(* CODESYS project pwm_01.project

Project tree, tasks and I/O mapping:
  Device : MC4-26-20, Enovation Controls, order no. 58-70-0006, version 1.1.0.17
      input  batteryVoltage : Word  // Battery Voltage
      input  reg1Voltage : Word  // Regulator #1 Voltage
      input  reg2Voltage : Word  // Regulator #2 Voltage
      input  wakePinVoltage : Word  // Wake Pin Voltage
      input  sleepAllowed : BIT  // Sleep Allowed
      output enterSleep : BIT  // Enter Sleep
      input  bootReason : Byte  // Bootup Reason
      output userLED1State : BIT  // User LED 1 State
      output userLED2State : BIT  // User LED 2 State
      input  loadpwrVoltage : Word  // Load Power Voltage
      input  loadpwrProtected : Word  // Load Power Voltage (Protected)
      input  topRailTemp : Int  // Top Heatrail Temp
      input  botRailTemp : Int  // Bottom Heatrail Temp
      input  buildMajorVersion : BYTE  // Build Major Version
      input  buildMinorVersion : BYTE  // Build Minor Version
      input  buildPatchVersion : BYTE  // Build Patch Version
      input  firmwareMajorVersion : DWord  // Firmware Major Version
      input  firmwareMinorVersion : DWord  // Firmware Minor Version
      input  firmwareIdentifier : DWord  // Firmware Identifier
      input  serialNumber : DWord  // Serial Number
      input  hourMeter : Real  // Hour Meter
      input  startCount : DWord  // Cumulative Starts
      input  dynamicMemSize : UINT  // Dynamic Memory Size
      input  dynamicMemMaxUsage : UINT  // Dynamic Memory Max Usage
      input  relayCurrent : Real  // Relay Total Current
      input  relaySourcing : Real  // Relay Sourcing Current
      input  relaySinking : Real  // Relay Sinking Current
      output relayState : BIT  // Relay State
      input  relayIsActive : BIT  // Relay Active
      output clearActiveFaults : BIT  // Clear Active Faults (rising edge)
      input  activeFaultIsSet : BIT  // Active Fault Available
      input  activeFaultCount : UINT  // Active Fault Count
      output clearHistoricFaults : BIT  // Clear Historic Faults (rising edge)
      input  historicFaultIsSet : BIT  // Historic Fault Available
      input  historicFaultCount : UINT  // Historic Fault Count
      input  totalFaultCount : UINT  // Total Fault Count
      output fltMonIndex : UINT  // Fault Index
      input  fltMonIsEnabled : BIT  // Fault Is Enabled
      input  fltMonConditionPresent : BIT  // Fault Condition Present
      input  fltMonActive : BIT  // Fault Active Latched
      input  fltMonHistoric : BIT  // Fault Historic Latched
      input  fltMonCurrentStart : BIT  // Current start cycle
      input  fltMonActiveStarts : BYTE  // Starts since active
      output fltMonClearActive : BIT  // Clear Active (rising edge)
      output fltMonClearHistoric : BIT  // Clear Historic (rising edge)
      input  dcSwitchTemp : Int  // DC Switch Temp
      input  InputA04 : input_param_hi_spd_struct  // Input A04
      input  analogValueA04 : Real  // Input A04.Analog value
      input  digitalValueA04 : Bool  // Input A04.Digital value
      input  frequencyA04 : Word  // Input A04.Frequency
      input  dutyCycleA04 : Real  // Input A04.Duty cycle
      input  phaseAngleA04 : Real  // Input A04.Phase angle
      input  pulseCountA04 : DWord  // Input A04.Pulse count
      input  upDownCountA04 : DInt  // Input A04.Up/Down count
      input  freqHPA04 : Real  // Input A04.Frequency (high precision)
      input  freqTSA04 : Real  // Input A04.Frequency edge timestamp
      input  InputA05 : input_param_hi_spd_struct  // Input A05
      input  analogValueA05 : Real  // Input A05.Analog value
      input  digitalValueA05 : Bool  // Input A05.Digital value
      input  frequencyA05 : Word  // Input A05.Frequency
      input  dutyCycleA05 : Real  // Input A05.Duty cycle
      input  phaseAngleA05 : Real  // Input A05.Phase angle
      input  pulseCountA05 : DWord  // Input A05.Pulse count
      input  upDownCountA05 : DInt  // Input A05.Up/Down count
      input  freqHPA05 : Real  // Input A05.Frequency (high precision)
      input  freqTSA05 : Real  // Input A05.Frequency edge timestamp
      input  InputA07 : input_param_hi_spd_struct  // Input A07
      input  analogValueA07 : Real  // Input A07.Analog value
      input  digitalValueA07 : Bool  // Input A07.Digital value
      input  frequencyA07 : Word  // Input A07.Frequency
      input  dutyCycleA07 : Real  // Input A07.Duty cycle
      input  phaseAngleA07 : Real  // Input A07.Phase angle
      input  pulseCountA07 : DWord  // Input A07.Pulse count
      input  upDownCountA07 : DInt  // Input A07.Up/Down count
      input  freqHPA07 : Real  // Input A07.Frequency (high precision)
      input  freqTSA07 : Real  // Input A07.Frequency edge timestamp
      input  InputA10 : input_param_hi_spd_struct  // Input A10
      input  analogValueA10 : Real  // Input A10.Analog value
      input  digitalValueA10 : Bool  // Input A10.Digital value
      input  frequencyA10 : Word  // Input A10.Frequency
      input  dutyCycleA10 : Real  // Input A10.Duty cycle
      input  phaseAngleA10 : Real  // Input A10.Phase angle
      input  pulseCountA10 : DWord  // Input A10.Pulse count
      input  upDownCountA10 : DInt  // Input A10.Up/Down count
      input  freqHPA10 : Real  // Input A10.Frequency (high precision)
      input  freqTSA10 : Real  // Input A10.Frequency edge timestamp
      input  InputA11 : input_param_hi_spd_struct  // Input A11
      input  analogValueA11 : Real  // Input A11.Analog value
      input  digitalValueA11 : Bool  // Input A11.Digital value
      input  frequencyA11 : Word  // Input A11.Frequency
      input  dutyCycleA11 : Real  // Input A11.Duty cycle
      input  phaseAngleA11 : Real  // Input A11.Phase angle
      input  pulseCountA11 : DWord  // Input A11.Pulse count
      input  upDownCountyA11 : DInt  // Input A11.Up/Down count
      input  freqHPA11 : Real  // Input A11.Frequency (high precision)
      input  freqTSA11 : Real  // Input A11.Frequency edge timestamp
      input  InputA12 : input_param_hi_spd_struct  // Input A12
      input  analogValueA12 : Real  // Input A12.Analog value
      input  digitalValueA12 : Bool  // Input A12.Digital value
      input  frequencyA12 : Word  // Input A12.Frequency
      input  dutyCycleA12 : Real  // Input A12.Duty cycle
      input  phaseAngleA12 : Real  // Input A12.Phase angle
      input  pulseCountA12 : DWord  // Input A12.Pulse count
      input  upDownCountA12 : DInt  // Input A12.Up/Down count
      input  freqHPA12 : Real  // Input A12.Frequency (high precision)
      input  freqTSA12 : Real  // Input A12.Frequency edge timestamp
      input  InputB07 : input_param_hi_spd_struct  // Input B07
      input  analogValueB07 : Real  // Input B07.Analog value
      input  digitalValueB07 : Bool  // Input B07.Digital value
      input  frequencyB07 : Word  // Input B07.Frequency
      input  dutyCycleB07 : Real  // Input B07.Duty cycle
      input  phaseAngleB07 : Real  // Input B07.Phase angle
      input  pulseCountB07 : DWord  // Input B07.Pulse count
      input  upDownCountB07 : DInt  // Input B07.Up/Down count
      input  freqHPB07 : Real  // Input B07.Frequency (high precision)
      input  freqTSB07 : Real  // Input B07.Frequency edge timestamp
      input  InputB08 : input_param_hi_spd_struct  // Input B08
      input  analogValueB08 : Real  // Input B08.Analog value
      input  digitalValueB08 : Bool  // Input B08.Digital value
      input  frequencyB08 : Word  // Input B08.Frequency
      input  dutyCycleB08 : Real  // Input B08.Duty cycle
      input  phaseAngleB08 : Real  // Input B08.Phase angle
      input  pulseCountB08 : DWord  // Input B08.Pulse count
      input  upDownCountB08 : DInt  // Input B08.Up/Down count
      input  freqHPB08 : Real  // Input B08.Frequency (high precision)
      input  freqTSB08 : Real  // Input B08.Frequency edge timestamp
      input  InputB09 : input_param_hi_spd_struct  // Input B09
      input  analogValueB09 : Real  // Input B09.Analog value
      input  digitalValueB09 : Bool  // Input B09.Digital value
      input  frequencyB09 : Word  // Input B09.Frequency
      input  dutyCycleB09 : Real  // Input B09.Duty cycle
      input  phaseAngleB09 : Real  // Input B09.Phase angle
      input  pulseCountB09 : DWord  // Input B09.Pulse count
      input  upDownCountB09 : DInt  // Input B09.Up/Down count
      input  freqHPB09 : Real  // Input B09.Frequency (high precision)
      input  freqTSB09 : Real  // Input B09.Frequency edge timestamp
      input  InputB10 : input_param_hi_spd_struct  // Input B10
      input  analogValueB10 : Real  // Input B10.Analog value
      input  digitalValueB10 : Bool  // Input B10.Digital value
      input  frequencyB10 : Word  // Input B10.Frequency
      input  dutyCycleB10 : Real  // Input B10.Duty cycle
      input  phaseAngleB10 : Real  // Input B10.Phase angle
      input  pulseCountB10 : DWord  // Input B10.Pulse count
      input  upDownCountB10 : DInt  // Input B10.Up/Down count
      input  freqHPB10 : Real  // Input B10.Frequency (high precision)
      input  freqTSB10 : Real  // Input B10.Frequency edge timestamp
      input  InputA06 : input_param_struct  // Input A06
      input  analogValueA06 : Real  // Input A06.Analog value
      input  digitalValueA06 : Bool  // Input A06.Digital value
      input  frequencyA06 : Word  // Input A06.Frequency
      input  pulseCountA06 : DWord  // Input A06.Pulse count
      input  freqHPA06 : Real  // Input A06.Frequency (high precision)
      input  freqTSA06 : Real  // Input A06.Frequency edge timestamp
      input  InputA14 : input_param_struct  // Input A14
      input  analogValueA14 : Real  // Input A14.Analog value
      input  digitalValueA14 : Bool  // Input A14.Digital value
      input  frequencyA14 : Word  // Input A14.Frequency
      input  pulseCountA14 : DWord  // Input A14.Pulse count
      input  freqHPA14 : Real  // Input A14.Frequency (high precision)
      input  freqTSA14 : Real  // Input A14.Frequency edge timestamp
      input  InputA15 : input_param_struct  // Input A15
      input  analogValueA15 : Real  // Input A15.Analog value
      input  digitalValueA15 : Bool  // Input A15.Digital value
      input  frequencyA15 : Word  // Input A15.Frequency
      input  pulseCountA15 : DWord  // Input A15.Pulse count
      input  freqHPA15 : Real  // Input A15.Frequency (high precision)
      input  freqTSA15 : Real  // Input A15.Frequency edge timestamp
      input  InputA16 : input_param_struct  // Input A16
      input  analogValueA16 : Real  // Input A16.Analog value
      input  digitalValueA16 : Bool  // Input A16.Digital value
      input  frequencyA16 : Word  // Input A16.Frequency
      input  pulseCountA16 : DWord  // Input A16.Pulse count
      input  freqHPA16 : Real  // Input A16.Frequency (high precision)
      input  freqTSA16 : Real  // Input A16.Frequency edge timestamp
      input  InputA17 : input_param_struct  // Input A17
      input  analogValueA17 : Real  // Input A17.Analog value
      input  digitalValueA17 : Bool  // Input A17.Digital value
      input  frequencyA17 : Word  // Input A17.Frequency
      input  pulseCountA17 : DWord  // Input A17.Pulse count
      input  freqHPA17 : Real  // Input A17.Frequency (high precision)
      input  freqTSA17 : Real  // Input A17.Frequency edge timestamp
      input  InputA18 : input_param_struct  // Input A18
      input  analogValueA18 : Real  // Input A18.Analog value
      input  digitalValueA18 : Bool  // Input A18.Digital value
      input  frequencyA18 : Word  // Input A18.Frequency
      input  pulseCountA18 : DWord  // Input A18.Pulse count
      input  freqHPA18 : Real  // Input A18.Frequency (high precision)
      input  freqTSA18 : Real  // Input A18.Frequency edge timestamp
      input  InputB01 : input_param_struct  // Input B01
      input  analogValueB01 : Real  // Input B01.Analog value
      input  digitalValueB01 : Bool  // Input B01.Digital value
      input  frequencyB01 : Word  // Input B01.Frequency
      input  pulseCountB01 : DWord  // Input B01.Pulse count
      input  freqHPB01 : Real  // Input B01.Frequency (high precision)
      input  freqTSB01 : Real  // Input B01.Frequency edge timestamp
      input  InputB11 : input_param_struct  // Input B11
      input  analogValueB11 : Real  // Input B11.Analog value
      input  digitalValueB11 : Bool  // Input B11.Digital value
      input  frequencyB11 : Word  // Input B11.Frequency
      input  pulseCountB11 : DWord  // Input B11.Pulse count
      input  freqHPB11 : Real  // Input B11.Frequency (high precision)
      input  freqTSB11 : Real  // Input B11.Frequency edge timestamp
      input  InputB12 : input_param_struct  // Input B12
      input  analogValueB12 : Real  // Input B12.Analog value
      input  digitalValueB12 : Bool  // Input B12.Digital value
      input  frequencyB12 : Word  // Input B12.Frequency
      input  pulseCountB12 : DWord  // Input B12.Pulse count
      input  freqHPB12 : Real  // Input B12.Frequency (high precision)
      input  freqTSB12 : Real  // Input B12.Frequency edge timestamp
      input  InputB13 : input_param_struct  // Input B13
      input  analogValueB13 : Real  // Input B13.Analog value
      input  digitalValueB13 : Bool  // Input B13.Digital value
      input  frequencyB13 : Word  // Input B13.Frequency
      input  pulseCountB13 : DWord  // Input B13.Pulse count
      input  freqHPB13 : Real  // Input B13.Frequency (high precision)
      input  freqTSB13 : Real  // Input B13.Frequency edge timestamp
      input  InputC07 : input_param_struct  // Input C07
      input  analogValueC07 : Real  // Input C07.Analog value
      input  digitalValueC07 : Bool  // Input C07.Digital value
      input  frequencyC07 : Word  // Input C07.Frequency
      input  pulseCountC07 : DWord  // Input C07.Pulse count
      input  freqHPC07 : Real  // Input C07.Frequency (high precision)
      input  freqTSC07 : Real  // Input C07.Frequency edge timestamp
      input  InputC08 : input_param_struct  // Input C08
      input  analogValueC08 : Real  // Input C08.Analog value
      input  digitalValueC08 : Bool  // Input C08.Digital value
      input  frequencyC08 : Word  // Input C08.Frequency
      input  pulseCountC08 : DWord  // Input C08.Pulse count
      input  freqHPC08 : Real  // Input C08.Frequency (high precision)
      input  freqTSC08 : Real  // Input C08.Frequency edge timestamp
      input  InputC09 : input_param_struct  // Input C09
      input  analogValueC09 : Real  // Input C09.Analog value
      input  digitalValueC09 : Bool  // Input C09.Digital value
      input  frequencyC09 : Word  // Input C09.Frequency
      input  pulseCountC09 : DWord  // Input C09.Pulse count
      input  freqHPC09 : Real  // Input C09.Frequency (high precision)
      input  freqTSC09 : Real  // Input C09.Frequency edge timestamp
      input  InputC10 : input_param_struct  // Input C10
      input  analogValueC10 : Real  // Input C10.Analog value
      input  digitalValueC10 : Bool  // Input C10.Digital value
      input  frequencyC10 : Word  // Input C10.Frequency
      input  pulseCountC10 : DWord  // Input C10.Pulse count
      input  freqHPC10 : Real  // Input C10.Frequency (high precision)
      input  freqTSC10 : Real  // Input C10.Frequency edge timestamp
      input  InputC11 : input_param_struct  // Input C11
      input  analogValueC11 : Real  // Input C11.Analog value
      input  digitalValueC11 : Bool  // Input C11.Digital value
      input  frequencyC11 : Word  // Input C11.Frequency
      input  pulseCountC11 : DWord  // Input C11.Pulse count
      input  freqHPC11 : Real  // Input C11.Frequency (high precision)
      input  freqTSC11 : Real  // Input C11.Frequency edge timestamp
      input  InputC12 : input_param_struct  // Input C12
      input  analogValueC12 : Real  // Input C12.Analog value
      input  digitalValueC12 : Bool  // Input C12.Digital value
      input  frequencyC12 : Word  // Input C12.Frequency
      input  pulseCountC12 : DWord  // Input C12.Pulse count
      input  freqHPC12 : Real  // Input C12.Frequency (high precision)
      input  freqTSC12 : Real  // Input C12.Frequency edge timestamp
      input  chanStateB02 : Byte  // Channel state
      input  chanStateB03 : Byte  // Channel state
      input  chanStateB04 : Byte  // Channel state
      input  chanStateB05 : Byte  // Channel state
      input  chanStateB06 : Byte  // Channel state
      input  chanStateB14 : Byte  // Channel state
      input  chanStateB15 : Byte  // Channel state
      input  chanStateB16 : Byte  // Channel state
      input  chanStateB17 : Byte  // Channel state
      input  chanStateB18 : Byte  // Channel state
      input  chanStateC02 : Byte  // Channel state
      input  chanStateC03 : Byte  // Channel state
      input  chanStateC04 : Byte  // Channel state
      input  chanStateC05 : Byte  // Channel state
      input  chanStateC06 : Byte  // Channel state
      input  chanStateC14 : Byte  // Channel state
      input  chanStateC15 : Byte  // Channel state
      input  chanStateC16 : Byte  // Channel state
      input  chanStateC17 : Byte  // Channel state
      input  chanStateC18 : Byte  // Channel state
      output desiredDutyB02 : Real  // Desired Duty Cycle
      output desiredDutyB03 : Real  // Desired Duty Cycle
      output desiredDutyB04 : Real  // Desired Duty Cycle
      output desiredDutyB05 : Real  // Desired Duty Cycle
      output desiredDutyB06 : Real  // Desired Duty Cycle
      output desiredDutyB14 : Real  // Desired Duty Cycle
      output desiredDutyB15 : Real  // Desired Duty Cycle
      output desiredDutyB16 : Real  // Desired Duty Cycle
      output desiredDutyB17 : Real  // Desired Duty Cycle
      output desiredDutyB18 : Real  // Desired Duty Cycle
      output desiredDutyC02 : Real  // Desired Duty Cycle
      output desiredDutyC03 : Real  // Desired Duty Cycle
      output desiredDutyC04 : Real  // Desired Duty Cycle
      output desiredDutyC05 : Real  // Desired Duty Cycle
      output desiredDutyC06 : Real  // Desired Duty Cycle
      output desiredDutyC14 : Real  // Desired Duty Cycle
      output desiredDutyC15 : Real  // Desired Duty Cycle
      output desiredDutyC16 : Real  // Desired Duty Cycle
      output desiredDutyC17 : Real  // Desired Duty Cycle
      output desiredDutyC18 : Real  // Desired Duty Cycle
      input  actualDutyB02 : Real  // Actual Duty Cycle
      input  actualDutyB03 : Real  // Actual Duty Cycle
      input  actualDutyB04 : Real  // Actual Duty Cycle
      input  actualDutyB05 : Real  // Actual Duty Cycle
      input  actualDutyB06 : Real  // Actual Duty Cycle
      input  actualDutyB14 : Real  // Actual Duty Cycle
      input  actualDutyB15 : Real  // Actual Duty Cycle
      input  actualDutyB16 : Real  // Actual Duty Cycle
      input  actualDutyB17 : Real  // Actual Duty Cycle
      input  actualDutyB18 : Real  // Actual Duty Cycle
      input  actualDutyC02 : Real  // Actual Duty Cycle
      input  actualDutyC03 : Real  // Actual Duty Cycle
      input  actualDutyC04 : Real  // Actual Duty Cycle
      input  actualDutyC05 : Real  // Actual Duty Cycle
      input  actualDutyC06 : Real  // Actual Duty Cycle
      input  actualDutyC14 : Real  // Actual Duty Cycle
      input  actualDutyC15 : Real  // Actual Duty Cycle
      input  actualDutyC16 : Real  // Actual Duty Cycle
      input  actualDutyC17 : Real  // Actual Duty Cycle
      input  actualDutyC18 : Real  // Actual Duty Cycle
      output desiredCurrentB02 : Real  // Desired Current
      output desiredCurrentB03 : Real  // Desired Current
      output desiredCurrentB04 : Real  // Desired Current
      output desiredCurrentB05 : Real  // Desired Current
      output desiredCurrentB06 : Real  // Desired Current
      output desiredCurrentB14 : Real  // Desired Current
      output desiredCurrentB15 : Real  // Desired Current
      output desiredCurrentB16 : Real  // Desired Current
      output desiredCurrentB17 : Real  // Desired Current
      output desiredCurrentB18 : Real  // Desired Current
      output desiredCurrentC02 : Real  // Desired Current
      output desiredCurrentC03 : Real  // Desired Current
      output desiredCurrentC04 : Real  // Desired Current
      output desiredCurrentC05 : Real  // Desired Current
      output desiredCurrentC06 : Real  // Desired Current
      output desiredCurrentC14 : Real  // Desired Current
      output desiredCurrentC15 : Real  // Desired Current
      output desiredCurrentC16 : Real  // Desired Current
      output desiredCurrentC17 : Real  // Desired Current
      output desiredCurrentC18 : Real  // Desired Current
      input  measuredCurrentB02 : Real  // Current Feedback
      input  measuredCurrentB03 : Real  // Current Feedback
      input  measuredCurrentB04 : Real  // Current Feedback
      input  measuredCurrentB05 : Real  // Current Feedback
      input  measuredCurrentB06 : Real  // Current Feedback
      input  measuredCurrentB14 : Real  // Current Feedback
      input  measuredCurrentB15 : Real  // Current Feedback
      input  measuredCurrentB16 : Real  // Current Feedback
      input  measuredCurrentB17 : Real  // Current Feedback
      input  measuredCurrentB18 : Real  // Current Feedback
      input  measuredCurrentC02 : Real  // Current Feedback
      input  measuredCurrentC03 : Real  // Current Feedback
      input  measuredCurrentC04 : Real  // Current Feedback
      input  measuredCurrentC05 : Real  // Current Feedback
      input  measuredCurrentC06 : Real  // Current Feedback
      input  measuredCurrentC14 : Real  // Current Feedback
      input  measuredCurrentC15 : Real  // Current Feedback
      input  measuredCurrentC16 : Real  // Current Feedback
      input  measuredCurrentC17 : Real  // Current Feedback
      input  measuredCurrentC18 : Real  // Current Feedback
      output binaryOutputB02 : BIT  // Digital Output
      output binaryOutputB03 : BIT  // Digital Output
      output binaryOutputB04 : BIT  // Digital Output
      output binaryOutputB05 : BIT  // Digital Output
      output binaryOutputB06 : BIT  // Digital Output
      output binaryOutputB14 : BIT  // Digital Output
      output binaryOutputB15 : BIT  // Digital Output
      output binaryOutputB16 : BIT  // Digital Output
      output binaryOutputB17 : BIT  // Digital Output
      output binaryOutputB18 : BIT  // Digital Output
      output binaryOutputC02 : BIT  // Digital Output
      output binaryOutputC03 : BIT  // Digital Output
      output binaryOutputC04 : BIT  // Digital Output
      output binaryOutputC05 : BIT  // Digital Output
      output binaryOutputC06 : BIT  // Digital Output
      output binaryOutputC14 : BIT  // Digital Output
      output binaryOutputC15 : BIT  // Digital Output
      output binaryOutputC16 : BIT  // Digital Output
      output binaryOutputC17 : BIT  // Digital Output
      output binaryOutputC18 : BIT  // Digital Output
      output hbridgeActionB02 : Byte  // H-Bridge Action
      output hbridgeActionB03 : Byte  // H-Bridge Action
      output hbridgeActionB04 : Byte  // H-Bridge Action
      output hbridgeActionB05 : Byte  // H-Bridge Action
      output hbridgeActionB06 : Byte  // H-Bridge Action
      output hbridgeActionB14 : Byte  // H-Bridge Action
      output hbridgeActionB15 : Byte  // H-Bridge Action
      output hbridgeActionB16 : Byte  // H-Bridge Action
      output hbridgeActionB17 : Byte  // H-Bridge Action
      output hbridgeActionB18 : Byte  // H-Bridge Action
      output hbridgeActionC02 : Byte  // H-Bridge Action
      output hbridgeActionC03 : Byte  // H-Bridge Action
      output hbridgeActionC04 : Byte  // H-Bridge Action
      output hbridgeActionC05 : Byte  // H-Bridge Action
      output hbridgeActionC06 : Byte  // H-Bridge Action
      output hbridgeActionC14 : Byte  // H-Bridge Action
      output hbridgeActionC15 : Byte  // H-Bridge Action
      output hbridgeActionC16 : Byte  // H-Bridge Action
      output hbridgeActionC17 : Byte  // H-Bridge Action
      output hbridgeActionC18 : Byte  // H-Bridge Action
      input  measuredVoltageB02 : Real  // Measured Voltage
      input  measuredVoltageB03 : Real  // Measured Voltage
      input  measuredVoltageB04 : Real  // Measured Voltage
      input  measuredVoltageB05 : Real  // Measured Voltage
      input  measuredVoltageB06 : Real  // Measured Voltage
      input  measuredVoltageB14 : Real  // Measured Voltage
      input  measuredVoltageB15 : Real  // Measured Voltage
      input  measuredVoltageB16 : Real  // Measured Voltage
      input  measuredVoltageB17 : Real  // Measured Voltage
      input  measuredVoltageB18 : Real  // Measured Voltage
      input  measuredVoltageC02 : Real  // Measured Voltage
      input  measuredVoltageC03 : Real  // Measured Voltage
      input  measuredVoltageC04 : Real  // Measured Voltage
      input  measuredVoltageC05 : Real  // Measured Voltage
      input  measuredVoltageC06 : Real  // Measured Voltage
      input  measuredVoltageC14 : Real  // Measured Voltage
      input  measuredVoltageC15 : Real  // Measured Voltage
      input  measuredVoltageC16 : Real  // Measured Voltage
      input  measuredVoltageC17 : Real  // Measured Voltage
      input  measuredVoltageC18 : Real  // Measured Voltage
      output setUserFaults : ARRAY[0..15] of BYTE  // 
      input  userFaultIsHistoric : ARRAY[0..15] of BYTE  // 
      input  systemFaultIsActive : ARRAY[0..60] of BYTE  // 
      input  systemFaultIsHistoric : ARRAY[0..60] of BYTE  // 
      unmapped channels: Active Fault IDs, Historic Fault IDs
    application Application
      libraries: Standard, 3.5.18.0 (System)
      task MainTask (cyclic, interval t#1000ms, priority 16) calls High_Side_Output
      program High_Side_Output [ST]
    System Config
        input  batteryVoltage : Word  // Battery Voltage
        input  reg1Voltage : Word  // Regulator #1 Voltage
        input  reg2Voltage : Word  // Regulator #2 Voltage
        input  wakePinVoltage : Word  // Wake Pin Voltage
        input  sleepAllowed : BIT  // Sleep Allowed
        output enterSleep : BIT  // Enter Sleep
        input  bootReason : Byte  // Bootup Reason
        output userLED1State : BIT  // User LED 1 State
        output userLED2State : BIT  // User LED 2 State
        input  loadpwrVoltage : Word  // Load Power Voltage
        input  loadpwrProtected : Word  // Load Power Voltage (Protected)
        input  topRailTemp : Int  // Top Heatrail Temp
        input  botRailTemp : Int  // Bottom Heatrail Temp
        input  buildMajorVersion : BYTE  // Build Major Version
        input  buildMinorVersion : BYTE  // Build Minor Version
        input  buildPatchVersion : BYTE  // Build Patch Version
        input  firmwareMajorVersion : DWord  // Firmware Major Version
        input  firmwareMinorVersion : DWord  // Firmware Minor Version
        input  firmwareIdentifier : DWord  // Firmware Identifier
        input  serialNumber : DWord  // Serial Number
        input  hourMeter : Real  // Hour Meter
        input  startCount : DWord  // Cumulative Starts
        input  dynamicMemSize : UINT  // Dynamic Memory Size
        input  dynamicMemMaxUsage : UINT  // Dynamic Memory Max Usage
        input  relayCurrent : Real  // Relay Total Current
        input  relaySourcing : Real  // Relay Sourcing Current
        input  relaySinking : Real  // Relay Sinking Current
        output relayState : BIT  // Relay State
        input  relayIsActive : BIT  // Relay Active
        output clearActiveFaults : BIT  // Clear Active Faults (rising edge)
        input  activeFaultIsSet : BIT  // Active Fault Available
        input  activeFaultCount : UINT  // Active Fault Count
        output clearHistoricFaults : BIT  // Clear Historic Faults (rising edge)
        input  historicFaultIsSet : BIT  // Historic Fault Available
        input  historicFaultCount : UINT  // Historic Fault Count
        input  totalFaultCount : UINT  // Total Fault Count
        output fltMonIndex : UINT  // Fault Index
        input  fltMonIsEnabled : BIT  // Fault Is Enabled
        input  fltMonConditionPresent : BIT  // Fault Condition Present
        input  fltMonActive : BIT  // Fault Active Latched
        input  fltMonHistoric : BIT  // Fault Historic Latched
        input  fltMonCurrentStart : BIT  // Current start cycle
        input  fltMonActiveStarts : BYTE  // Starts since active
        output fltMonClearActive : BIT  // Clear Active (rising edge)
        output fltMonClearHistoric : BIT  // Clear Historic (rising edge)
        input  dcSwitchTemp : Int  // DC Switch Temp
        unmapped channels: Active Fault IDs, Historic Fault IDs
    Inputs
        input  InputA04 : input_param_hi_spd_struct  // Input A04
        input  analogValueA04 : Real  // Input A04.Analog value
        input  digitalValueA04 : Bool  // Input A04.Digital value
        input  frequencyA04 : Word  // Input A04.Frequency
        input  dutyCycleA04 : Real  // Input A04.Duty cycle
        input  phaseAngleA04 : Real  // Input A04.Phase angle
        input  pulseCountA04 : DWord  // Input A04.Pulse count
        input  upDownCountA04 : DInt  // Input A04.Up/Down count
        input  freqHPA04 : Real  // Input A04.Frequency (high precision)
        input  freqTSA04 : Real  // Input A04.Frequency edge timestamp
        input  InputA05 : input_param_hi_spd_struct  // Input A05
        input  analogValueA05 : Real  // Input A05.Analog value
        input  digitalValueA05 : Bool  // Input A05.Digital value
        input  frequencyA05 : Word  // Input A05.Frequency
        input  dutyCycleA05 : Real  // Input A05.Duty cycle
        input  phaseAngleA05 : Real  // Input A05.Phase angle
        input  pulseCountA05 : DWord  // Input A05.Pulse count
        input  upDownCountA05 : DInt  // Input A05.Up/Down count
        input  freqHPA05 : Real  // Input A05.Frequency (high precision)
        input  freqTSA05 : Real  // Input A05.Frequency edge timestamp
        input  InputA07 : input_param_hi_spd_struct  // Input A07
        input  analogValueA07 : Real  // Input A07.Analog value
        input  digitalValueA07 : Bool  // Input A07.Digital value
        input  frequencyA07 : Word  // Input A07.Frequency
        input  dutyCycleA07 : Real  // Input A07.Duty cycle
        input  phaseAngleA07 : Real  // Input A07.Phase angle
        input  pulseCountA07 : DWord  // Input A07.Pulse count
        input  upDownCountA07 : DInt  // Input A07.Up/Down count
        input  freqHPA07 : Real  // Input A07.Frequency (high precision)
        input  freqTSA07 : Real  // Input A07.Frequency edge timestamp
        input  InputA10 : input_param_hi_spd_struct  // Input A10
        input  analogValueA10 : Real  // Input A10.Analog value
        input  digitalValueA10 : Bool  // Input A10.Digital value
        input  frequencyA10 : Word  // Input A10.Frequency
        input  dutyCycleA10 : Real  // Input A10.Duty cycle
        input  phaseAngleA10 : Real  // Input A10.Phase angle
        input  pulseCountA10 : DWord  // Input A10.Pulse count
        input  upDownCountA10 : DInt  // Input A10.Up/Down count
        input  freqHPA10 : Real  // Input A10.Frequency (high precision)
        input  freqTSA10 : Real  // Input A10.Frequency edge timestamp
        input  InputA11 : input_param_hi_spd_struct  // Input A11
        input  analogValueA11 : Real  // Input A11.Analog value
        input  digitalValueA11 : Bool  // Input A11.Digital value
        input  frequencyA11 : Word  // Input A11.Frequency
        input  dutyCycleA11 : Real  // Input A11.Duty cycle
        input  phaseAngleA11 : Real  // Input A11.Phase angle
        input  pulseCountA11 : DWord  // Input A11.Pulse count
        input  upDownCountyA11 : DInt  // Input A11.Up/Down count
        input  freqHPA11 : Real  // Input A11.Frequency (high precision)
        input  freqTSA11 : Real  // Input A11.Frequency edge timestamp
        input  InputA12 : input_param_hi_spd_struct  // Input A12
        input  analogValueA12 : Real  // Input A12.Analog value
        input  digitalValueA12 : Bool  // Input A12.Digital value
        input  frequencyA12 : Word  // Input A12.Frequency
        input  dutyCycleA12 : Real  // Input A12.Duty cycle
        input  phaseAngleA12 : Real  // Input A12.Phase angle
        input  pulseCountA12 : DWord  // Input A12.Pulse count
        input  upDownCountA12 : DInt  // Input A12.Up/Down count
        input  freqHPA12 : Real  // Input A12.Frequency (high precision)
        input  freqTSA12 : Real  // Input A12.Frequency edge timestamp
        input  InputB07 : input_param_hi_spd_struct  // Input B07
        input  analogValueB07 : Real  // Input B07.Analog value
        input  digitalValueB07 : Bool  // Input B07.Digital value
        input  frequencyB07 : Word  // Input B07.Frequency
        input  dutyCycleB07 : Real  // Input B07.Duty cycle
        input  phaseAngleB07 : Real  // Input B07.Phase angle
        input  pulseCountB07 : DWord  // Input B07.Pulse count
        input  upDownCountB07 : DInt  // Input B07.Up/Down count
        input  freqHPB07 : Real  // Input B07.Frequency (high precision)
        input  freqTSB07 : Real  // Input B07.Frequency edge timestamp
        input  InputB08 : input_param_hi_spd_struct  // Input B08
        input  analogValueB08 : Real  // Input B08.Analog value
        input  digitalValueB08 : Bool  // Input B08.Digital value
        input  frequencyB08 : Word  // Input B08.Frequency
        input  dutyCycleB08 : Real  // Input B08.Duty cycle
        input  phaseAngleB08 : Real  // Input B08.Phase angle
        input  pulseCountB08 : DWord  // Input B08.Pulse count
        input  upDownCountB08 : DInt  // Input B08.Up/Down count
        input  freqHPB08 : Real  // Input B08.Frequency (high precision)
        input  freqTSB08 : Real  // Input B08.Frequency edge timestamp
        input  InputB09 : input_param_hi_spd_struct  // Input B09
        input  analogValueB09 : Real  // Input B09.Analog value
        input  digitalValueB09 : Bool  // Input B09.Digital value
        input  frequencyB09 : Word  // Input B09.Frequency
        input  dutyCycleB09 : Real  // Input B09.Duty cycle
        input  phaseAngleB09 : Real  // Input B09.Phase angle
        input  pulseCountB09 : DWord  // Input B09.Pulse count
        input  upDownCountB09 : DInt  // Input B09.Up/Down count
        input  freqHPB09 : Real  // Input B09.Frequency (high precision)
        input  freqTSB09 : Real  // Input B09.Frequency edge timestamp
        input  InputB10 : input_param_hi_spd_struct  // Input B10
        input  analogValueB10 : Real  // Input B10.Analog value
        input  digitalValueB10 : Bool  // Input B10.Digital value
        input  frequencyB10 : Word  // Input B10.Frequency
        input  dutyCycleB10 : Real  // Input B10.Duty cycle
        input  phaseAngleB10 : Real  // Input B10.Phase angle
        input  pulseCountB10 : DWord  // Input B10.Pulse count
        input  upDownCountB10 : DInt  // Input B10.Up/Down count
        input  freqHPB10 : Real  // Input B10.Frequency (high precision)
        input  freqTSB10 : Real  // Input B10.Frequency edge timestamp
        input  InputA06 : input_param_struct  // Input A06
        input  analogValueA06 : Real  // Input A06.Analog value
        input  digitalValueA06 : Bool  // Input A06.Digital value
        input  frequencyA06 : Word  // Input A06.Frequency
        input  pulseCountA06 : DWord  // Input A06.Pulse count
        input  freqHPA06 : Real  // Input A06.Frequency (high precision)
        input  freqTSA06 : Real  // Input A06.Frequency edge timestamp
        input  InputA14 : input_param_struct  // Input A14
        input  analogValueA14 : Real  // Input A14.Analog value
        input  digitalValueA14 : Bool  // Input A14.Digital value
        input  frequencyA14 : Word  // Input A14.Frequency
        input  pulseCountA14 : DWord  // Input A14.Pulse count
        input  freqHPA14 : Real  // Input A14.Frequency (high precision)
        input  freqTSA14 : Real  // Input A14.Frequency edge timestamp
        input  InputA15 : input_param_struct  // Input A15
        input  analogValueA15 : Real  // Input A15.Analog value
        input  digitalValueA15 : Bool  // Input A15.Digital value
        input  frequencyA15 : Word  // Input A15.Frequency
        input  pulseCountA15 : DWord  // Input A15.Pulse count
        input  freqHPA15 : Real  // Input A15.Frequency (high precision)
        input  freqTSA15 : Real  // Input A15.Frequency edge timestamp
        input  InputA16 : input_param_struct  // Input A16
        input  analogValueA16 : Real  // Input A16.Analog value
        input  digitalValueA16 : Bool  // Input A16.Digital value
        input  frequencyA16 : Word  // Input A16.Frequency
        input  pulseCountA16 : DWord  // Input A16.Pulse count
        input  freqHPA16 : Real  // Input A16.Frequency (high precision)
        input  freqTSA16 : Real  // Input A16.Frequency edge timestamp
        input  InputA17 : input_param_struct  // Input A17
        input  analogValueA17 : Real  // Input A17.Analog value
        input  digitalValueA17 : Bool  // Input A17.Digital value
        input  frequencyA17 : Word  // Input A17.Frequency
        input  pulseCountA17 : DWord  // Input A17.Pulse count
        input  freqHPA17 : Real  // Input A17.Frequency (high precision)
        input  freqTSA17 : Real  // Input A17.Frequency edge timestamp
        input  InputA18 : input_param_struct  // Input A18
        input  analogValueA18 : Real  // Input A18.Analog value
        input  digitalValueA18 : Bool  // Input A18.Digital value
        input  frequencyA18 : Word  // Input A18.Frequency
        input  pulseCountA18 : DWord  // Input A18.Pulse count
        input  freqHPA18 : Real  // Input A18.Frequency (high precision)
        input  freqTSA18 : Real  // Input A18.Frequency edge timestamp
        input  InputB01 : input_param_struct  // Input B01
        input  analogValueB01 : Real  // Input B01.Analog value
        input  digitalValueB01 : Bool  // Input B01.Digital value
        input  frequencyB01 : Word  // Input B01.Frequency
        input  pulseCountB01 : DWord  // Input B01.Pulse count
        input  freqHPB01 : Real  // Input B01.Frequency (high precision)
        input  freqTSB01 : Real  // Input B01.Frequency edge timestamp
        input  InputB11 : input_param_struct  // Input B11
        input  analogValueB11 : Real  // Input B11.Analog value
        input  digitalValueB11 : Bool  // Input B11.Digital value
        input  frequencyB11 : Word  // Input B11.Frequency
        input  pulseCountB11 : DWord  // Input B11.Pulse count
        input  freqHPB11 : Real  // Input B11.Frequency (high precision)
        input  freqTSB11 : Real  // Input B11.Frequency edge timestamp
        input  InputB12 : input_param_struct  // Input B12
        input  analogValueB12 : Real  // Input B12.Analog value
        input  digitalValueB12 : Bool  // Input B12.Digital value
        input  frequencyB12 : Word  // Input B12.Frequency
        input  pulseCountB12 : DWord  // Input B12.Pulse count
        input  freqHPB12 : Real  // Input B12.Frequency (high precision)
        input  freqTSB12 : Real  // Input B12.Frequency edge timestamp
        input  InputB13 : input_param_struct  // Input B13
        input  analogValueB13 : Real  // Input B13.Analog value
        input  digitalValueB13 : Bool  // Input B13.Digital value
        input  frequencyB13 : Word  // Input B13.Frequency
        input  pulseCountB13 : DWord  // Input B13.Pulse count
        input  freqHPB13 : Real  // Input B13.Frequency (high precision)
        input  freqTSB13 : Real  // Input B13.Frequency edge timestamp
        input  InputC07 : input_param_struct  // Input C07
        input  analogValueC07 : Real  // Input C07.Analog value
        input  digitalValueC07 : Bool  // Input C07.Digital value
        input  frequencyC07 : Word  // Input C07.Frequency
        input  pulseCountC07 : DWord  // Input C07.Pulse count
        input  freqHPC07 : Real  // Input C07.Frequency (high precision)
        input  freqTSC07 : Real  // Input C07.Frequency edge timestamp
        input  InputC08 : input_param_struct  // Input C08
        input  analogValueC08 : Real  // Input C08.Analog value
        input  digitalValueC08 : Bool  // Input C08.Digital value
        input  frequencyC08 : Word  // Input C08.Frequency
        input  pulseCountC08 : DWord  // Input C08.Pulse count
        input  freqHPC08 : Real  // Input C08.Frequency (high precision)
        input  freqTSC08 : Real  // Input C08.Frequency edge timestamp
        input  InputC09 : input_param_struct  // Input C09
        input  analogValueC09 : Real  // Input C09.Analog value
        input  digitalValueC09 : Bool  // Input C09.Digital value
        input  frequencyC09 : Word  // Input C09.Frequency
        input  pulseCountC09 : DWord  // Input C09.Pulse count
        input  freqHPC09 : Real  // Input C09.Frequency (high precision)
        input  freqTSC09 : Real  // Input C09.Frequency edge timestamp
        input  InputC10 : input_param_struct  // Input C10
        input  analogValueC10 : Real  // Input C10.Analog value
        input  digitalValueC10 : Bool  // Input C10.Digital value
        input  frequencyC10 : Word  // Input C10.Frequency
        input  pulseCountC10 : DWord  // Input C10.Pulse count
        input  freqHPC10 : Real  // Input C10.Frequency (high precision)
        input  freqTSC10 : Real  // Input C10.Frequency edge timestamp
        input  InputC11 : input_param_struct  // Input C11
        input  analogValueC11 : Real  // Input C11.Analog value
        input  digitalValueC11 : Bool  // Input C11.Digital value
        input  frequencyC11 : Word  // Input C11.Frequency
        input  pulseCountC11 : DWord  // Input C11.Pulse count
        input  freqHPC11 : Real  // Input C11.Frequency (high precision)
        input  freqTSC11 : Real  // Input C11.Frequency edge timestamp
        input  InputC12 : input_param_struct  // Input C12
        input  analogValueC12 : Real  // Input C12.Analog value
        input  digitalValueC12 : Bool  // Input C12.Digital value
        input  frequencyC12 : Word  // Input C12.Frequency
        input  pulseCountC12 : DWord  // Input C12.Pulse count
        input  freqHPC12 : Real  // Input C12.Frequency (high precision)
        input  freqTSC12 : Real  // Input C12.Frequency edge timestamp
    Outputs
        input  chanStateB02 : Byte  // Channel state
        input  chanStateB03 : Byte  // Channel state
        input  chanStateB04 : Byte  // Channel state
        input  chanStateB05 : Byte  // Channel state
        input  chanStateB06 : Byte  // Channel state
        input  chanStateB14 : Byte  // Channel state
        input  chanStateB15 : Byte  // Channel state
        input  chanStateB16 : Byte  // Channel state
        input  chanStateB17 : Byte  // Channel state
        input  chanStateB18 : Byte  // Channel state
        input  chanStateC02 : Byte  // Channel state
        input  chanStateC03 : Byte  // Channel state
        input  chanStateC04 : Byte  // Channel state
        input  chanStateC05 : Byte  // Channel state
        input  chanStateC06 : Byte  // Channel state
        input  chanStateC14 : Byte  // Channel state
        input  chanStateC15 : Byte  // Channel state
        input  chanStateC16 : Byte  // Channel state
        input  chanStateC17 : Byte  // Channel state
        input  chanStateC18 : Byte  // Channel state
        output desiredDutyB02 : Real  // Desired Duty Cycle
        output desiredDutyB03 : Real  // Desired Duty Cycle
        output desiredDutyB04 : Real  // Desired Duty Cycle
        output desiredDutyB05 : Real  // Desired Duty Cycle
        output desiredDutyB06 : Real  // Desired Duty Cycle
        output desiredDutyB14 : Real  // Desired Duty Cycle
        output desiredDutyB15 : Real  // Desired Duty Cycle
        output desiredDutyB16 : Real  // Desired Duty Cycle
        output desiredDutyB17 : Real  // Desired Duty Cycle
        output desiredDutyB18 : Real  // Desired Duty Cycle
        output desiredDutyC02 : Real  // Desired Duty Cycle
        output desiredDutyC03 : Real  // Desired Duty Cycle
        output desiredDutyC04 : Real  // Desired Duty Cycle
        output desiredDutyC05 : Real  // Desired Duty Cycle
        output desiredDutyC06 : Real  // Desired Duty Cycle
        output desiredDutyC14 : Real  // Desired Duty Cycle
        output desiredDutyC15 : Real  // Desired Duty Cycle
        output desiredDutyC16 : Real  // Desired Duty Cycle
        output desiredDutyC17 : Real  // Desired Duty Cycle
        output desiredDutyC18 : Real  // Desired Duty Cycle
        input  actualDutyB02 : Real  // Actual Duty Cycle
        input  actualDutyB03 : Real  // Actual Duty Cycle
        input  actualDutyB04 : Real  // Actual Duty Cycle
        input  actualDutyB05 : Real  // Actual Duty Cycle
        input  actualDutyB06 : Real  // Actual Duty Cycle
        input  actualDutyB14 : Real  // Actual Duty Cycle
        input  actualDutyB15 : Real  // Actual Duty Cycle
        input  actualDutyB16 : Real  // Actual Duty Cycle
        input  actualDutyB17 : Real  // Actual Duty Cycle
        input  actualDutyB18 : Real  // Actual Duty Cycle
        input  actualDutyC02 : Real  // Actual Duty Cycle
        input  actualDutyC03 : Real  // Actual Duty Cycle
        input  actualDutyC04 : Real  // Actual Duty Cycle
        input  actualDutyC05 : Real  // Actual Duty Cycle
        input  actualDutyC06 : Real  // Actual Duty Cycle
        input  actualDutyC14 : Real  // Actual Duty Cycle
        input  actualDutyC15 : Real  // Actual Duty Cycle
        input  actualDutyC16 : Real  // Actual Duty Cycle
        input  actualDutyC17 : Real  // Actual Duty Cycle
        input  actualDutyC18 : Real  // Actual Duty Cycle
        output desiredCurrentB02 : Real  // Desired Current
        output desiredCurrentB03 : Real  // Desired Current
        output desiredCurrentB04 : Real  // Desired Current
        output desiredCurrentB05 : Real  // Desired Current
        output desiredCurrentB06 : Real  // Desired Current
        output desiredCurrentB14 : Real  // Desired Current
        output desiredCurrentB15 : Real  // Desired Current
        output desiredCurrentB16 : Real  // Desired Current
        output desiredCurrentB17 : Real  // Desired Current
        output desiredCurrentB18 : Real  // Desired Current
        output desiredCurrentC02 : Real  // Desired Current
        output desiredCurrentC03 : Real  // Desired Current
        output desiredCurrentC04 : Real  // Desired Current
        output desiredCurrentC05 : Real  // Desired Current
        output desiredCurrentC06 : Real  // Desired Current
        output desiredCurrentC14 : Real  // Desired Current
        output desiredCurrentC15 : Real  // Desired Current
        output desiredCurrentC16 : Real  // Desired Current
        output desiredCurrentC17 : Real  // Desired Current
        output desiredCurrentC18 : Real  // Desired Current
        input  measuredCurrentB02 : Real  // Current Feedback
        input  measuredCurrentB03 : Real  // Current Feedback
        input  measuredCurrentB04 : Real  // Current Feedback
        input  measuredCurrentB05 : Real  // Current Feedback
        input  measuredCurrentB06 : Real  // Current Feedback
        input  measuredCurrentB14 : Real  // Current Feedback
        input  measuredCurrentB15 : Real  // Current Feedback
        input  measuredCurrentB16 : Real  // Current Feedback
        input  measuredCurrentB17 : Real  // Current Feedback
        input  measuredCurrentB18 : Real  // Current Feedback
        input  measuredCurrentC02 : Real  // Current Feedback
        input  measuredCurrentC03 : Real  // Current Feedback
        input  measuredCurrentC04 : Real  // Current Feedback
        input  measuredCurrentC05 : Real  // Current Feedback
        input  measuredCurrentC06 : Real  // Current Feedback
        input  measuredCurrentC14 : Real  // Current Feedback
        input  measuredCurrentC15 : Real  // Current Feedback
        input  measuredCurrentC16 : Real  // Current Feedback
        input  measuredCurrentC17 : Real  // Current Feedback
        input  measuredCurrentC18 : Real  // Current Feedback
        output binaryOutputB02 : BIT  // Digital Output
        output binaryOutputB03 : BIT  // Digital Output
        output binaryOutputB04 : BIT  // Digital Output
        output binaryOutputB05 : BIT  // Digital Output
        output binaryOutputB06 : BIT  // Digital Output
        output binaryOutputB14 : BIT  // Digital Output
        output binaryOutputB15 : BIT  // Digital Output
        output binaryOutputB16 : BIT  // Digital Output
        output binaryOutputB17 : BIT  // Digital Output
        output binaryOutputB18 : BIT  // Digital Output
        output binaryOutputC02 : BIT  // Digital Output
        output binaryOutputC03 : BIT  // Digital Output
        output binaryOutputC04 : BIT  // Digital Output
        output binaryOutputC05 : BIT  // Digital Output
        output binaryOutputC06 : BIT  // Digital Output
        output binaryOutputC14 : BIT  // Digital Output
        output binaryOutputC15 : BIT  // Digital Output
        output binaryOutputC16 : BIT  // Digital Output
        output binaryOutputC17 : BIT  // Digital Output
        output binaryOutputC18 : BIT  // Digital Output
        output hbridgeActionB02 : Byte  // H-Bridge Action
        output hbridgeActionB03 : Byte  // H-Bridge Action
        output hbridgeActionB04 : Byte  // H-Bridge Action
        output hbridgeActionB05 : Byte  // H-Bridge Action
        output hbridgeActionB06 : Byte  // H-Bridge Action
        output hbridgeActionB14 : Byte  // H-Bridge Action
        output hbridgeActionB15 : Byte  // H-Bridge Action
        output hbridgeActionB16 : Byte  // H-Bridge Action
        output hbridgeActionB17 : Byte  // H-Bridge Action
        output hbridgeActionB18 : Byte  // H-Bridge Action
        output hbridgeActionC02 : Byte  // H-Bridge Action
        output hbridgeActionC03 : Byte  // H-Bridge Action
        output hbridgeActionC04 : Byte  // H-Bridge Action
        output hbridgeActionC05 : Byte  // H-Bridge Action
        output hbridgeActionC06 : Byte  // H-Bridge Action
        output hbridgeActionC14 : Byte  // H-Bridge Action
        output hbridgeActionC15 : Byte  // H-Bridge Action
        output hbridgeActionC16 : Byte  // H-Bridge Action
        output hbridgeActionC17 : Byte  // H-Bridge Action
        output hbridgeActionC18 : Byte  // H-Bridge Action
        input  measuredVoltageB02 : Real  // Measured Voltage
        input  measuredVoltageB03 : Real  // Measured Voltage
        input  measuredVoltageB04 : Real  // Measured Voltage
        input  measuredVoltageB05 : Real  // Measured Voltage
        input  measuredVoltageB06 : Real  // Measured Voltage
        input  measuredVoltageB14 : Real  // Measured Voltage
        input  measuredVoltageB15 : Real  // Measured Voltage
        input  measuredVoltageB16 : Real  // Measured Voltage
        input  measuredVoltageB17 : Real  // Measured Voltage
        input  measuredVoltageB18 : Real  // Measured Voltage
        input  measuredVoltageC02 : Real  // Measured Voltage
        input  measuredVoltageC03 : Real  // Measured Voltage
        input  measuredVoltageC04 : Real  // Measured Voltage
        input  measuredVoltageC05 : Real  // Measured Voltage
        input  measuredVoltageC06 : Real  // Measured Voltage
        input  measuredVoltageC14 : Real  // Measured Voltage
        input  measuredVoltageC15 : Real  // Measured Voltage
        input  measuredVoltageC16 : Real  // Measured Voltage
        input  measuredVoltageC17 : Real  // Measured Voltage
        input  measuredVoltageC18 : Real  // Measured Voltage
    Fault Table
        output setUserFaults : ARRAY[0..15] of BYTE  // 
        input  userFaultIsHistoric : ARRAY[0..15] of BYTE  // 
        input  systemFaultIsActive : ARRAY[0..60] of BYTE  // 
        input  systemFaultIsHistoric : ARRAY[0..60] of BYTE  // 
*)

// Device/Application/High_Side_Output
PROGRAM High_Side_Output
VAR
	counter     : UINT  := 0;
	LED1state   : BOOL := FALSE;
	LED2state   : BOOL := FALSE;

END_VAR

VAR CONSTANT
	ON 			: BOOL := TRUE;
	OFF 		: BOOL := FALSE;
	
END_VAR

// STEP 1: Always turn on the Solid State Relay to enable all PWM Outputs
// STEP 2: Configure Output Configurtaion B02 Drive Profile = Single, Drive Mode = PWM, Switching Side = HS
// STEP 3: Set the desired duty cycle of the output


// Enable the Solid State Relay 
IF IoConfig_Globals_Mapping.relayState = FALSE THEN
	IoConfig_Globals_Mapping.relayState := TRUE;
END_IF

// Toggle Output B02 between On/Off each pass through the loop
//Mirror the state of the output on user LED #1

LED1state :=IoConfig_Globals_Mapping.userLed1State;

IF LED1state = OFF THEN
	LED1state := ON;
//turn output ON with PWM of 50%
	desiredDutyB02 := 50;
	IoConfig_Globals_Mapping.userLed1State := TRUE;

ELSE 
	LED1state := OFF;
//Turn output OFF with PWM of 0%
	desiredDutyB02 := 0;
	IoConfig_Globals_Mapping.userLed1State := FALSE;
END_IF

END_PROGRAM
